// TIA Portal V18 export
FUNCTION_BLOCK "MU_Spin"   // FB31, LAD
TITLE = MU Spin
{ S7_Optimized_Access := 'TRUE' }
// Written BY Kristopher Gimenez Feb 3,2023
// This block is used to control the TD MU Spin mode
// stored: AutoNumber false, MemoryReserve 100, SetENOAutomatically false
   VAR_OUTPUT
      FlowFwdmAOut : Real;
      TorqmAOut : Real;
      FwdEnableP1 : Bool;
      FwdEnableP2 : Bool;
      TorqEn : Bool;
   END_VAR
   VAR
      LinkExtSw_Last : Bool;
      LinkRetSw_Last : Bool;
      MUSpinComplete : Bool;
   END_VAR
   VAR_TEMP
      TorqPSITemp : Real;
   END_VAR
   VAR_TEMP   // added for the SCL form of the ladder/FBD networks
      _w1 : Bool;
      _w2 : Bool;
      _w3 : Bool;
   END_VAR
BEGIN

REGION Network 1: Speed Adjust
   // If PTO confirmed in MU Spin mode allow user to adjust spin speed setpoint using Link Tilt Joysticks
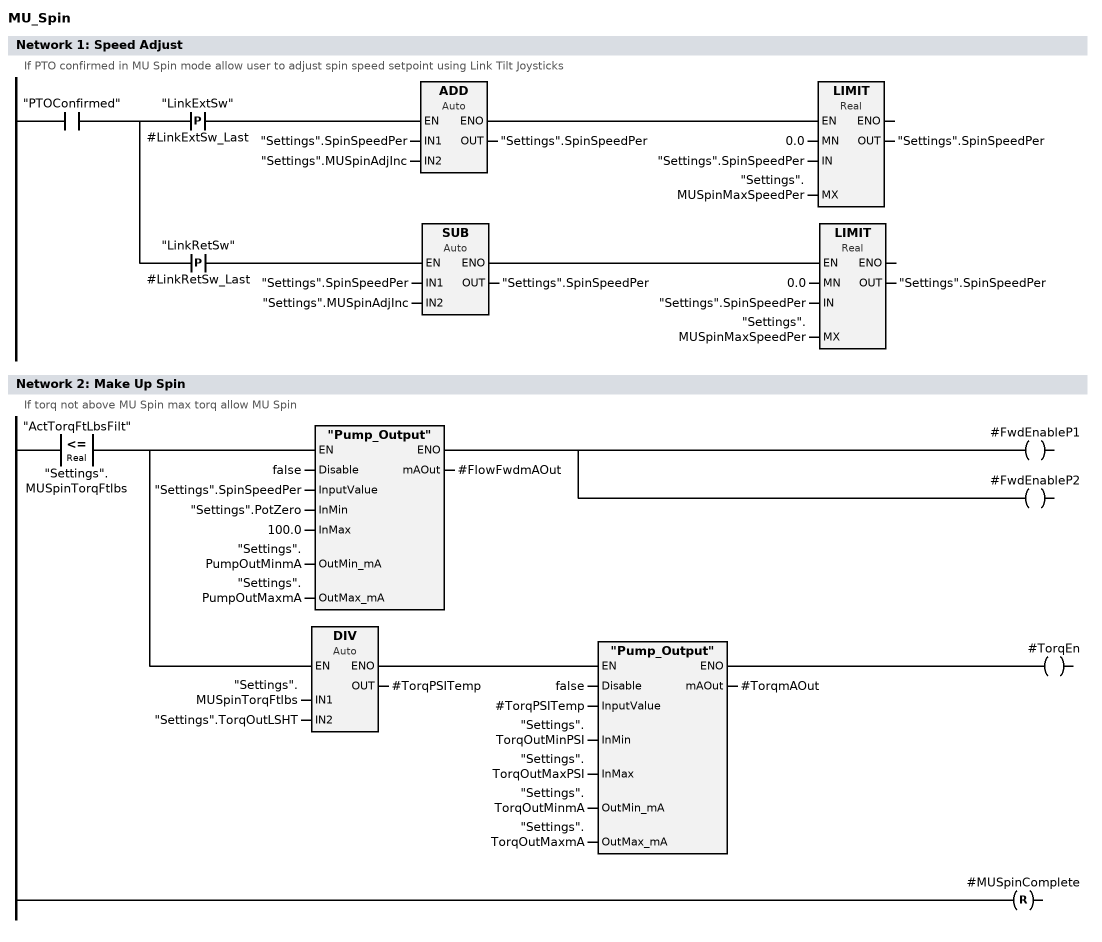
   RUNG wire#powerrail
      Contact( "PTOConfirmed" )
      wire#w1
      P_Contact(operand := "LinkExtSw", bit := #LinkExtSw_Last)
      Add(in1 := "Settings".SpinSpeedPer, in2 := "Settings".MUSpinAdjInc, out => "Settings".SpinSpeedPer)
      { S7_Templates := "value_type := Real" } Limit(mn := 0.0, in := "Settings".SpinSpeedPer, mx := "Settings".MUSpinMaxSpeedPer, out => "Settings".SpinSpeedPer)
   END_RUNG
   RUNG wire#w1
      P_Contact(operand := "LinkRetSw", bit := #LinkRetSw_Last)
      Sub(in1 := "Settings".SpinSpeedPer, in2 := "Settings".MUSpinAdjInc, out => "Settings".SpinSpeedPer)
      { S7_Templates := "value_type := Real" } Limit(mn := 0.0, in := "Settings".SpinSpeedPer, mx := "Settings".MUSpinMaxSpeedPer, out => "Settings".SpinSpeedPer)
   END_RUNG
   // the same network as SCL:
   #_w1 := "PTOConfirmed" AND "LinkExtSw" AND NOT #LinkExtSw_Last;   // rising edge of "LinkExtSw"
   #LinkExtSw_Last := "LinkExtSw";
   IF #_w1 THEN
       "Settings".SpinSpeedPer := "Settings".SpinSpeedPer + "Settings".MUSpinAdjInc;
       "Settings".SpinSpeedPer := LIMIT(MN := 0.0, IN := "Settings".SpinSpeedPer, MX := "Settings".MUSpinMaxSpeedPer);
   END_IF;
   #_w2 := "PTOConfirmed" AND "LinkRetSw" AND NOT #LinkRetSw_Last;   // rising edge of "LinkRetSw"
   #LinkRetSw_Last := "LinkRetSw";
   IF #_w2 THEN
       "Settings".SpinSpeedPer := "Settings".SpinSpeedPer - "Settings".MUSpinAdjInc;
       "Settings".SpinSpeedPer := LIMIT(MN := 0.0, IN := "Settings".SpinSpeedPer, MX := "Settings".MUSpinMaxSpeedPer);
   END_IF;
END_REGION

REGION Network 2: Make Up Spin
   // If torq not above MU Spin max torq allow MU Spin
   RUNG wire#powerrail
      { S7_Templates := "SrcType := Real" } LE_Contact(in1 := "ActTorqFtLbsFilt", in2 := "Settings".MUSpinTorqFtlbs)
      wire#w1
      "Pump_Output"(Disable := false, InputValue := "Settings".SpinSpeedPer, InMin := "Settings".PotZero, InMax := 100.0, OutMin_mA := "Settings".PumpOutMinmA, OutMax_mA := "Settings".PumpOutMaxmA, mAOut => #FlowFwdmAOut)
      wire#w2
      Coil( #FwdEnableP1 )
   END_RUNG
   RUNG wire#w2
      Coil( #FwdEnableP2 )
   END_RUNG
   RUNG wire#w1
      Div(in1 := "Settings".MUSpinTorqFtlbs, in2 := "Settings".TorqOutLSHT, out => #TorqPSITemp)
      "Pump_Output"(Disable := false, InputValue := #TorqPSITemp, InMin := "Settings".TorqOutMinPSI, InMax := "Settings".TorqOutMaxPSI, OutMin_mA := "Settings".TorqOutMinmA, OutMax_mA := "Settings".TorqOutMaxmA, mAOut => #TorqmAOut)
      Coil( #TorqEn )
   END_RUNG
   RUNG wire#powerrail
      R_Coil( #MUSpinComplete )
   END_RUNG
   // the same network as SCL:
   #_w2 := "ActTorqFtLbsFilt" <= "Settings".MUSpinTorqFtlbs;
   "Pump_Output"(EN := "ActTorqFtLbsFilt" <= "Settings".MUSpinTorqFtlbs,
                 Disable := false,
                 InputValue := "Settings".SpinSpeedPer,
                 InMin := "Settings".PotZero,
                 InMax := 100.0,
                 OutMin_mA := "Settings".PumpOutMinmA,
                 OutMax_mA := "Settings".PumpOutMaxmA,
                 mAOut => #FlowFwdmAOut,
                 ENO => #_w1);
   #FwdEnableP1 := #_w1;
   #FwdEnableP2 := #_w1;
   IF #_w2 THEN #TorqPSITemp := "Settings".MUSpinTorqFtlbs / "Settings".TorqOutLSHT; END_IF;
   "Pump_Output"(EN := #_w2,
                 Disable := false,
                 InputValue := #TorqPSITemp,
                 InMin := "Settings".TorqOutMinPSI,
                 InMax := "Settings".TorqOutMaxPSI,
                 OutMin_mA := "Settings".TorqOutMinmA,
                 OutMax_mA := "Settings".TorqOutMaxmA,
                 mAOut => #TorqmAOut,
                 ENO => #_w3);
   #TorqEn := #_w3;
   #MUSpinComplete := FALSE;
END_REGION
END_FUNCTION_BLOCK
